# EPICS substitutions: modules/event/evrSupport/Db/ioc/IOC-LI21-BP01bsa.substitutions
# BSA records
# One per device:
# Please check the HOPR,LOPR,PREC,ADEL,MDEL values provided in bsaBPMSEdef.db!
file bsaBPMSEdef.db {
#      Device        ,loc'n , IOC unit, timing system
  pattern {DEVICE    , LOC  ,  UN  , SYS  , SLCLNK}
	  { BPMS:LI21:131, LI21 , BP01 , SYS0 , BPMS:LI21:131:FANOUTSLC}
	  { BPMS:LI21:161, LI21 , BP01 , SYS0 , BPMS:LI21:161:FANOUTSLC}
	  { BPMS:LI21:201, LI21 , BP01 , SYS0 , BPMS:LI21:201:FANOUTSLC}
	  { BPMS:LI21:233, LI21 , BP01 , SYS0 , BPMS:LI21:233:FANOUTSLC}
	  { BPMS:LI21:278, LI21 , BP01 , SYS0 , BPMS:LI21:278:FANOUTSLC}
	  { BPMS:LI21:301, LI21 , BP01 , SYS0 , BPMS:LI21:301:FANOUTSLC}
	  { BPMS:LI21:315, LI21 , BP01 , SYS0 , BPMS:LI21:315:FANOUTSLC}
}
